PROGRAM OP70_AUTOSEQUENCE
VAR
	OP70_Oring_OK 	: BOOL;
	FIXTURE_LH		: INT;
	FIXTURE_RH 		: INT;
	del : ton;
	tmp :BOOL;	
	Gripper_Delay: TON;
	Gripper_Aft_Place_Delay	: TON;
	Dry_Run : BOOL;
	OP70_STN_MOVER: INT;
	OP70_Cycle_Time_FB : FB_Cycletime;
	PAP_CYC_VAR : BOOL;
	OP70_PAP_Cycle_time : UDINT;
	OP70_Overall_Cyc_Time	: UDINT;
	OP70_PAP_Cycle_Time_FB : FB_Cycletime;
	OP70_Continous_Run : BOOL;
END_VAR

VAR PERSISTENT

END_VAR

// AUTO MODE
IF (NOT OP70_AutoSelected OR  OP70_ErrorActive OR OP70_HomeRunning ) THEN
	OP70_AutoRunning:= FALSE;
	OP70_Conveyor_ON:=FALSE;
	OP70_AutoSeq:= 10;
END_IF	

IF OP70_AutoSelected THEN
	OP70_GIUDE_GRP_ctrl.Position:=OP70_Guide_Pos;
	OP70_GIUDE_GRP_ctrl.Velocity:=50;	
	SR70_Vert_servo_ctrl.Velocity:=OP70_HMI_Servo_Speed_Vertical;
	SR70_HORI_servo_ctrl.Velocity:=OP70_HMI_Servo_Speed_Horizontal;	
END_IF

IF NOT OP70_AutoRunning THEN
    OP70_GIUDE_GRP_ctrl.Position:=0;
	OP70_GIUDE_GRP_ctrl.Velocity:=70;
	IF NOT In_Range(OP70_GIUDE_GRP_ctrl.Actual_Position,0,0.5) THEN
		OP70_GIUDE_GRP_ctrl.ABSmove_Start:=TRUE;
	END_IF	
END_IF

CASE OP70_AutoSeq OF
	    10: IF (OP70_AutoSelected) THEN		// Check Automode Selected
				OP70_AutoSeq:=20;
	        END_IF
		
	    20:IF ( NOT OP70_ErrorActive) THEN		//Check No error
		       OP70_AutoSeq:=30;
      	   END_IF
		   
      	30:IF (NOT OP70_HomeRunning) THEN		//Check No Homerunning
      		   OP70_AutoSeq :=40;
      	   END_IF
		   
        40:IF (OP70_Main.OP70_Modeselection_FB.TempHomeOK)THEN	//Check Machine in Home
      		   OP70_AutoSeq:= 50;
      	   END_IF
		   
      	50:IF ( NOT OP70_OperationCompleted) THEN		// Check Operation Completed Reset
      		   OP70_AutoSeq:=60;
      	   END_IF
		   
		60:IF  ( OP70_AutoRunning OR (NOT OP70_AutoRunning AND OP70_HMI_Cycle_Start )) THEN		//Machine Start in Fully Automatic or Press Cycle Start For Semi Automatic
		    OP70_GVL.OP70_HomeConditionOK:=TRUE;
	 			IF( OP70_Main.OP70_Modeselection_FB.HomeConditionOK AND OP70_AutoSelected) THEN
					OP70_GVL.OP70_AutoRunning:=TRUE;
					OP70_GVL.OP70_StepRunning:= FALSE;				
				ELSIF (OP70_Main.OP70_Modeselection_FB.HomeConditionOK AND OP70_StepSelected) THEN
					OP70_GVL.OP70_AutoRunning:=FALSE;
					OP70_GVL.OP70_StepRunning:= TRUE;
				END_IF;
		  END_IF
		   IF ((OP70_AutoRunning OR OP70_StepRunning) AND OP70_StartEnable) THEN
			   	OP70_GIUDE_GRP_ctrl.ABSmove_Start:=TRUE;
				OP70_Conveyor_ON:=TRUE;
				OP70_AutoSeq:= 65;
		   END_IF	
		   
		65 :  OP70_Gripper_LH_Close:=TRUE;  //CHECKING GRIPPER STATE BEFORE GRIPPING
			  OP70_Gripper_RH_Close:=TRUE;
			  IF NOT OP70_Gripper_LH_State AND NOT OP70_Gripper_RH_State THEN
				   OP70_AutoSeq:=66;
			  ELSE 	   
				   OP70_AutoSeq:=220;
			  END_IF 
			  
	    66: PAP_CYC_VAR:=1;
			IF OP70_pick_ready THEN
				OP70_AutoSeq:=70;
			ELSE 
				OP70_AutoSeq:=86;	
			END_IF 
		   
		70 : //MOVING HORIZONTAL SERVO TO PICK POSITION
			  IF (OP70_HORI_SERVO_ON_SFE_WRK_PICK OR OP70_HORI_SERVO_ON_SFE_WRK OR OP70_HORI_SERVO_ON_HOME OR OP70_HORI_SERVO_ON_WRK_PLACE OR OP70_HORI_SERVO_ON_WRK_PICK )AND OP70_HORI_SERVO_POS_DONE AND NOT SR70_HORI_servo_ctrl.ABSmove_Start THEN 
			   SR70_Hori_servo_ctrl.Position:=OP70_HORI_SERVO_PICK_POS;
               OP70_AutoSeq:=80; 			  
	          END_IF
			 
		80 :  SR70_HORI_servo_ctrl.ABSmove_Start := TRUE;     //HORIZONTAL SERVO MOVING
		       IF OP70_HORI_SERVO_ON_WRK_PICK THEN
				   SR70_HORI_servo_ctrl.ABSmove_Start := FALSE;
				   IF OP70_Gripper_LH_State AND OP70_Gripper_RH_State THEN
				        OP70_AutoSeq:=85;
				   ELSE 
						OP70_AutoSeq:=82;
				   END_IF
			   END_IF
		
	  	82 :  OP70_Gripper_LH_Close:=TRUE;  //CHECKING GRIPPER STATE BEFORE GRIPPING
			  OP70_Gripper_RH_Close:=TRUE;
			  IF NOT OP70_Gripper_LH_State AND NOT OP70_Gripper_RH_State THEN
				   OP70_AutoSeq:=85;
			  END_IF
			   
		85:	   // MOVING VERTICAL SERVO TO PICK POSITION
               IF  OP70_HORI_SERVO_ON_WRK_PICK AND (OP70_VERT_SERVO_ON_SFE_WRK OR OP70_VERT_SERVO_ON_HOME) AND 
				   OP70_VERT_SERVO_POS_DONE AND NOT SR70_VERT_servo_ctrl.ABSmove_Start  THEN
				   SR70_Vert_servo_ctrl.Position:=OP70_VERT_SERVO_PICK_POS;
				   SR70_VERT_servo_ctrl.ABSmove_Start := TRUE;
              	   OP70_AutoSeq:=100;			   
			   END_IF

	    86:   IF (OP70_HORI_SERVO_ON_SFE_WRK OR OP70_HORI_SERVO_ON_HOME OR OP70_HORI_SERVO_ON_WRK_PLACE OR OP70_HORI_SERVO_ON_WRK_PICK )AND OP70_HORI_SERVO_POS_DONE AND NOT SR70_HORI_servo_ctrl.ABSmove_Start THEN 
			    SR70_Hori_servo_ctrl.Position:=OP70_HORI_SERVO_SAFE_PICK_POS;
			    SR70_HORI_servo_ctrl.ABSmove_Start := TRUE;
                OP70_AutoSeq:=90;
			  END_IF
			   		  
		90 :  IF OP70_pick_ready THEN  // WAITING FOR O-RING TO BE OK AND THEN MOVING THE VERTICAL SERVO
			 		SR70_Hori_servo_ctrl.Position:=OP70_HORI_SERVO_PICK_POS;
					//SR70_Hori_servo_ctrl.ABSmove_Start := TRUE;
					OP70_AutoSeq:=92;
		      END_IF	
			  				
		92:  SR70_Hori_servo_ctrl.ABSmove_Start := TRUE;
			 IF OP70_HORI_SERVO_ON_WRK_PICK THEN
				 SR70_Vert_servo_ctrl.Position:=OP70_VERT_SERVO_PICK_POS;
				 SR70_VERT_servo_ctrl.ABSmove_Start := TRUE;
				 OP70_AutoSeq:=100;
			 END_IF 
	   
	   100 : IF OP70_VERT_SERVO_ON_WRK_PICK AND NOT SR70_VERT_servo_ctrl.ABSmove_Start THEN
				 SR70_VERT_servo_ctrl.ABSmove_Start := FALSE;
				 SR70_Vert_servo_ctrl.Position:=OP70_VERT_SERVO_SFE_WRK_POS; // FEEDING SAFE-WORK POSITION TO VERTICAL SERVO
              	 OP70_AutoSeq:=110;			   
			  END_IF	   
			 
      110:  IF NOT OP70_Grip_LH_Bypass THEN
				OP70_Gripper_LH_Open:=TRUE; 
			END_IF	
			IF NOT OP70_Grip_RH_Bypass THEN
    			OP70_Gripper_RH_Open:=TRUE;
			END_IF	
			IF Gripper_Delay.Q THEN
				 OP70_AutoSeq:=120;
		    END_IF
    		
      120: SR70_Hori_servo_ctrl.Position:=(OP70_HORI_SERVO_PICK_POS+OP70_Hori_Ser_Jerk_Pos);
	  	   SR70_HORI_servo_ctrl.ABSmove_Start := TRUE;
		   OP70_AutoSeq:=130;

    		   
      130:  SR70_HORI_servo_ctrl.ABSmove_Start := 0;
			SR70_VERT_servo_ctrl.ABSmove_Start := TRUE;	   //MOVING VERTICL SERVO TO SAFE-WORK
            IF OP70_VERT_SERVO_ON_SFE_WRK  THEN
    	      SR70_VERT_servo_ctrl.ABSmove_Start := FALSE;
			  OP70_pick_done:=TRUE;
              OP70_AutoSeq:=140;   
    		END_IF
    		   
      140:  IF (NOT OP70_Gripper_LH_State AND OP70_Grip_LH_Bypass ) AND OP70_Gripper_RH_State THEN  
    			OP70_AutoSeq:=150;
			ELSIF (NOT OP70_Gripper_RH_State AND OP70_Grip_RH_Bypass) AND OP70_Gripper_LH_State THEN
				OP70_AutoSeq:=150;
			ELSIF OP70_Gripper_LH_State AND OP70_Gripper_RH_State THEN  
    			OP70_AutoSeq:=150;
			ELSIF (NOT OP70_Gripper_LH_State AND NOT OP70_Grip_LH_Bypass) OR (NOT OP70_Gripper_RH_State AND NOT OP70_Grip_RH_Bypass) THEN	
				OP70_AutoSeq:=220;
			ELSIF OP70_Grip_LH_Bypass AND OP70_Grip_RH_Bypass THEN
				OP70_AutoSeq:=250;
			END_IF	
    	    		  
       150:  IF OP70_VERT_SERVO_ON_SFE_WRK  THEN // FEEDING PLACE POSITION TO HORIZONTAL SERVO
    		   SR70_Hori_servo_ctrl.Position:=OP70_HORI_SERVO_PLACE_POS;
               OP70_AutoSeq:=160;			 
    		 END_IF
    		   
       160:  SR70_HORI_servo_ctrl.ABSmove_Start := TRUE;    // MOVING HORIZONTAL SERVO TO PLACE POSITION
    		   IF OP70_HORI_SERVO_ON_WRK_PLACE THEN
    			 SR70_HORI_servo_ctrl.ABSmove_Start := FALSE;
    			 OP70_AutoSeq:=170;
    		   END_IF
       
       170: PAP_CYC_VAR:=0;
			IF OP70_HORI_SERVO_ON_WRK_PLACE AND NOT SR70_VERT_servo_ctrl.ABSmove_Start AND OP70_VERT_SERVO_ON_SFE_WRK AND OP70_STN_ENABLE THEN
    	   		SR70_Vert_servo_ctrl.Position:=OP70_VERT_SERVO_PLACE_POS;
              	OP70_AutoSeq:=175;	
      		END_IF
			
	   175: IF FIXTURE_LH<>60 AND FIXTURE_RH<>60 THEN
		   		OP70_AutoSeq:=250;	
			ELSIF FIXTURE_LH<>60 OR FIXTURE_RH<>60 THEN
				OP70_AutoSeq:=260;	
			ELSE
				OP70_AutoSeq:=180;		
	  	    END_IF			
    		
       180: SR70_VERT_servo_ctrl.ABSmove_Start := TRUE; //MOVING VERTICAL SERVO TO PLACE POSITION
    		IF OP70_VERT_SERVO_ON_WRK_PLACE THEN
    			SR70_VERT_servo_ctrl.ABSmove_Start := FALSE;
    			OP70_AutoSeq:=190;	
    		END_IF	
			
       190: IF FIXTURE_LH=60 AND NOT OP70_Grip_LH_Bypass THEN 
				OP70_Gripper_LH_Close:=TRUE;	
			END_IF	
			IF FIXTURE_RH=60 AND NOT OP70_Grip_RH_Bypass THEN 
				OP70_Gripper_RH_Close:=TRUE;	
			END_IF	
			tmp:=1;
			IF del.Q THEN		
				OP70_AutoSeq:=200;
			END_IF
			OP70_CURR_MOVER			:=OP70_STN_MOVER;
			
       200:  //MOVING BACK TO VERTICAL SERVO SAFE POSITION
    		 IF OP70_VERT_SERVO_ON_WRK_PLACE AND NOT SR70_VERT_servo_ctrl.ABSmove_Start THEN
    		   SR70_Vert_servo_ctrl.Position:=OP70_VERT_SERVO_SFE_WRK_POS;
               OP70_AutoSeq:=201;		   
    		 END_IF 

	   201: IF Dry_Run THEN
				OP70_AutoSeq:=210; 
			END_IF
			IF  FIXTURE_LH=60 AND FIXTURE_RH=60 THEN
				MOVER_CMP_STATUS[OP70_CURR_MOVER][1]:=70 ;
				MOVER_CMP_STATUS[OP70_CURR_MOVER][2]:=70 ;
				OP70_AutoSeq:=210;
			ELSIF FIXTURE_LH=60 THEN
				MOVER_CMP_STATUS[OP70_CURR_MOVER][1]:=70 ;
				OP70_AutoSeq:=210;
			ELSIF FIXTURE_RH=60 THEN
				MOVER_CMP_STATUS[OP70_CURR_MOVER][2]:=70 ;
				OP70_AutoSeq:=210;
			END_IF
    		 
       210:	 //PROCEEDING FOR NEXT CYCLE  
			  SR70_VERT_servo_ctrl.ABSmove_Start := TRUE;         
              IF OP70_VERT_SERVO_ON_SFE_WRK OR OP70_VERT_SERVO_ON_HOME  THEN
    			  SR70_VERT_servo_ctrl.ABSmove_Start := FALSE;
				  OP70_STN_ENABLE:=0;	  
    			  IF OP70_Gripper_LH_State OR OP70_Gripper_RH_State THEN
    		  		OP70_AutoSeq:=220;
    			  ELSIF (MOVER_CMP_STATUS[OP70_STN_MOVER][1]=70 OR MOVER_CMP_STATUS[OP70_STN_MOVER][2]=70) OR Dry_Run THEN
					STATION_DONE[OP70_CURR_MOVER][OP70_XTS_POS_NO]			:= TRUE;
					OP70_AutoSeq:=66;  
				  END_IF			  
    		  END_IF
    		  
       220:  IF (OP70_VERT_SERVO_ON_SFE_WRK OR OP70_VERT_SERVO_ON_HOME OR OP70_VERT_SERVO_ON_WRK_PLACE) AND NOT SR70_HORI_servo_ctrl.ABSmove_Start AND (OP70_HORI_SERVO_ON_WRK_PLACE OR OP70_HORI_SERVO_ON_WRK_Pick)  THEN
    		  SR70_Hori_servo_ctrl.Position:=OP70_HORI_SERVO_SFE_WRK_POS;
			  SR70_Vert_servo_ctrl.Position:=OP70_VERT_SERVO_SFE_WRK_POS;
			  SR70_VERT_servo_ctrl.ABSmove_Start := TRUE;
              OP70_AutoSeq:=240;			  
    		 END_IF  
    	
       240:  SR70_HORI_servo_ctrl.ABSmove_Start := TRUE;
             IF OP70_HORI_SERVO_ON_SFE_WRK THEN
    	  	   SR70_HORI_servo_ctrl.ABSmove_Start := FALSE;
      		   OP70_Gripper_RH_Close:=TRUE;	
    		   OP70_Gripper_LH_Close:=TRUE; 			   
      		 END_IF
    		 IF NOT OP70_Gripper_LH_State AND NOT OP70_Gripper_RH_State THEN
    		   OP70_AutoSeq:=66;
    		 END_IF
			 
		250://MOVER_CMP_STATUS[OP70_CURR_MOVER][1]:=71;
			//MOVER_CMP_STATUS[OP70_CURR_MOVER][2]:=71;
			OP70_STN_ENABLE:=0;	
			IF (MOVER_CMP_STATUS[OP70_STN_MOVER][1]=71 AND MOVER_CMP_STATUS[OP70_STN_MOVER][2]=71) THEN
				MOVER_STP_NO[OP70_CURR_MOVER]	:= (OP160_XTS_POS_NO*10);
			ELSE		
				STATION_DONE[OP70_CURR_MOVER][OP70_XTS_POS_NO]			:= TRUE;
			END_IF
				OP70_AutoSeq:=170; 	
	   260: SR70_Hori_servo_ctrl.Position:=OP70_HORI_SERVO_SFE_WRK_POS;
			SR70_Hori_servo_ctrl.ABSmove_Start:=TRUE;
			IF OP70_HORI_SERVO_ON_SFE_WRK THEN
				OP70_AutoSeq:=270; 
			END_IF
			
	   270: IF FIXTURE_LH<>60 AND NOT OP70_Grip_LH_Bypass THEN
				OP70_Gripper_LH_Close:=TRUE;
				IF NOT OP70_Gripper_LH_State THEN
					OP70_AutoSeq:=280; 
				END_IF
			ELSE
				OP70_AutoSeq:=280;	
			END_IF	
			
	   280: IF FIXTURE_RH<>60 AND NOT OP70_Grip_RH_Bypass THEN
				OP70_Gripper_RH_Close:=TRUE;
				IF NOT OP70_Gripper_RH_State THEN
					OP70_AutoSeq:=290; 
				END_IF
			ELSE
				OP70_AutoSeq:=290;	
			END_IF	

	   290: SR70_Hori_servo_ctrl.Position:=OP70_HORI_SERVO_PLACE_POS;
			SR70_Hori_servo_ctrl.ABSmove_Start:=TRUE;
			IF OP70_HORI_SERVO_ON_WRK_PLACE THEN
				OP70_AutoSeq:=180;	
			END_IF			 

END_CASE


OP70_STN_ENABLE:=OP70_Continous_Run;
				
OP70_Cycle_Time_FB(i_b_startTime:=OP70_STN_ENABLE , i_b_stopTime:= NOT OP70_STN_ENABLE , o_t_StationTime=>OP70_Cycle_time );					
OP70_PAP_Cycle_Time_FB(i_b_startTime:=PAP_CYC_VAR , i_b_stopTime:= NOT PAP_CYC_VAR , o_t_StationTime=>OP70_PAP_Cycle_time );					
OP70_Overall_Cyc_Time:=OP70_Cycle_time+OP70_PAP_Cycle_time;
	

Gripper_Delay(IN:=(OP70_AutoSeq=110),PT:=T#500MS);

Dry_Run:=All_Station_Dry_Run;
IF Dry_run THEN
	FIXTURE_LH :=60;	
    FIXTURE_RH :=60;
ELSE 
	FIXTURE_LH:=MOVER_CMP_STATUS[OP70_STN_MOVER][1];
	FIXTURE_RH:=MOVER_CMP_STATUS[OP70_STN_MOVER][2];	
END_IF	

del(IN:=tmp,PT:=T#700MS);
IF del.Q THEN
	tmp:=FALSE;
END_IF

// ################################			STATION ENABLE		####################################


OP70_STN_MOVER					:= MOVER_POSITION[OP70_XTS_POS_NO];

IF AUTO_WITH_XTS THEN
IF OP70_STN_MOVER>0 THEN
IF NOT(END_OF_CYCLE AND MOVER_CMP_STATUS[OP70_STN_MOVER][1]=5 AND MOVER_CMP_STATUS[OP70_STN_MOVER][2]=5)THEN	
	OP70_STN_ENABLE					:= MOVER_POS_RECHED[OP70_STN_MOVER] AND ((MOVER_CMP_STATUS[OP70_STN_MOVER][1]=60)OR
										(MOVER_CMP_STATUS[OP70_STN_MOVER][2]=60)) AND STATION_ENABLE_CONTROL;	
ELSE
	STATION_DONE[OP70_STN_MOVER][OP70_XTS_POS_NO]			:= TRUE;	
END_IF
ELSE
	OP70_STN_ENABLE					:= FALSE;
END_IF	
END_IF

END_PROGRAM

(* stored: Version 1.1.0.1, ProductVersion 3.1.4024.11
   POU OP70_AUTOSEQUENCE: Id {c3e594f8-85f7-4f1d-a499-aa1dfee21582}, SpecialFunc None *)
